// TIA Portal V20 export
FUNCTION "FC_AnalogInputsInit" : Void   // FC31, SCL
{ S7_Optimized_Access := 'TRUE' }
// stored: AutoNumber false, SetENOAutomatically false
   VAR_TEMP
      tBusy : Bool;
      tRetVal : Int;
   END_VAR
BEGIN
   REGION Description header 
       //==================================================================================
       // POSALUX Swiss SA / (C) Copyright 2025
       //----------------------------------------------------------------------------------
       // Title: Analog Inputs Initialisation 
       // Comment/Function: Initialisation of analog inputs
       // Author: Fabien WALDT
       // Engineering: TIA Portal v17
       //----------------------------------------------------------------------------------
       // Change log table:
       // Version  | Date     | Expert in charge | Changes applied
       // ---------|----------|------------------|-----------------------------------------
       // 00.00.01 | 20250423 | WFA              | First released version
       // =================================================================================
   END_REGION
   // Transfert Data From PLC to IHM at Start
   IF "FirstScan" THEN
       "DB_AnalogInputs".sLaserPowerMeter.sDownload := TRUE;
       "DB_AnalogInputs".sAxisB_ClampingPart.sDownload := TRUE;
       "DB_AnalogInputs".sLaserAirPressureProcess.sDownload := TRUE;
       "DB_AnalogInputs".sInletAirPressure.sDownload := TRUE;
       "DB_AnalogInputs".sAmbiantTemperature.sDownload := TRUE;
       "DB_AnalogInputs".sMachineTemperature.sDownload := TRUE;
       "DB_AnalogInputs".sCold_WaterTemperatureInput.sDownload := TRUE;
       "DB_AnalogInputs".sCold_WaterTemperatureOutput.sDownload := TRUE;
       "DB_AnalogInputs".sX_AxisTemperaturePT1000.sDownload := TRUE;
       "DB_AnalogInputs".sY_AxisTemperaturePT1000.sDownload := TRUE;
       "DB_AnalogInputs".sX_AxisTemperaturePTC.sDownload := TRUE;
       "DB_AnalogInputs".sY_AxisTemperaturePTC.sDownload := TRUE;
       "DB_AnalogInputs".sNozzleOverpressure.sDownload := TRUE;
       "DB_AnalogInputs".sOpticalPathOverpressure.sDownload := TRUE;
       "DB_AnalogInputs".sLaserHeadOverpressure.sDownload := TRUE;
       "DB_AnalogInputs".sZLAxisOverpressure.sDownload := TRUE;
       "DB_AnalogInputs".sXYAxisOverpressure.sDownload := TRUE;
       "DB_AnalogInputs".sLeftAspiration.sDownload := TRUE;
       "DB_AnalogInputs".sRightAspiration.sDownload := TRUE;
       "DB_AnalogInputs".sClimTemperature.sDownload := TRUE;
       "DB_AnalogInputs".sSensorControllerStation1.sDownload := TRUE;
       "DB_AnalogInputs".sCabinetTemperature.sDownload := TRUE;
   END_IF;

   // Update data from IHM
   IF "DB_OPC_AnalogInputs".Update THEN
       "DB_OPC_AnalogInputs".Signals["DB_OPC_AnalogInputs".Parameters.ItemNumber].Delay := LREAL_TO_REAL("DB_OPC_AnalogInputs".Parameters.Delay);
       "DB_OPC_AnalogInputs".Signals["DB_OPC_AnalogInputs".Parameters.ItemNumber].DiffErrorMax := LREAL_TO_REAL("DB_OPC_AnalogInputs".Parameters.DiffErrorMax);
       "DB_OPC_AnalogInputs".Signals["DB_OPC_AnalogInputs".Parameters.ItemNumber].DiffErrorMin := LREAL_TO_REAL("DB_OPC_AnalogInputs".Parameters.DiffErrorMin);
       "DB_OPC_AnalogInputs".Signals["DB_OPC_AnalogInputs".Parameters.ItemNumber].DiffWarnMax := LREAL_TO_REAL("DB_OPC_AnalogInputs".Parameters.DiffWarnMax);
       "DB_OPC_AnalogInputs".Signals["DB_OPC_AnalogInputs".Parameters.ItemNumber].DiffWarnMin := LREAL_TO_REAL("DB_OPC_AnalogInputs".Parameters.DiffWarnMin);
       "DB_OPC_AnalogInputs".Signals["DB_OPC_AnalogInputs".Parameters.ItemNumber].Id := DINT_TO_INT("DB_OPC_AnalogInputs".Parameters.Id);
       "DB_OPC_AnalogInputs".Signals["DB_OPC_AnalogInputs".Parameters.ItemNumber].Offset := LREAL_TO_REAL("DB_OPC_AnalogInputs".Parameters.Offset);
       "DB_OPC_AnalogInputs".Signals["DB_OPC_AnalogInputs".Parameters.ItemNumber].Gain := LREAL_TO_REAL("DB_OPC_AnalogInputs".Parameters.Gain);
       "DB_OPC_AnalogInputs".Signals["DB_OPC_AnalogInputs".Parameters.ItemNumber].Target := LREAL_TO_REAL("DB_OPC_AnalogInputs".Parameters.Target);

       "DB_OPC_AnalogInputs".Signals["DB_OPC_AnalogInputs".Parameters.ItemNumber].Update := TRUE;
       "DB_OPC_AnalogInputs".Update := FALSE;
   END_IF;

   // Permet de copier les valeurs en cours dans les valeurs initiales (A utiliser avec précautions)
   #tRetVal := WRIT_DBL(REQ := FALSE,
            SRCBLK := "DB_AnalogInputDataHMI",
            BUSY => #tBusy,
            DSTBLK => "DB_AnalogInputDataHMI");
END_FUNCTION
